TYPE M2TiltXAxisStatuses :
STRUCT
	///Is the axis healthy?
	healthStatus: HealthStatus;
END_STRUCT
END_TYPE

(* stored: Version 1.1.0.1, ProductVersion 3.1.4019.2
   DUT M2TiltXAxisStatuses: Id {5de5c23c-8e43-40ee-bcba-5b5e17c14200} *)
